FUNCTION_BLOCK FB_MotionInterlocksLimSw IMPLEMENTS I_MotionInterlocks
VAR_INPUT
END_VAR
VAR_OUTPUT
END_VAR
VAR
    iMotionInterlocksCommon : I_MotionInterlocksCommon;
    iLimSwStatus : I_LimSwStatus;
    bError : BOOL;
    nErrorID:UDINT;
    sMessage : T_MAXSTRING;
    {attribute 'hide'}
    bNewMoveReq : BOOL;
    {attribute 'hide'}
    bEnable	: BOOL;
    {attribute 'hide'}
    bReset : BOOL;
    {attribute 'hide'}
    bMoveOk : BOOL;
    bMoveBackwardEnabled : BOOL;
    bMoveForwardEnabled  : BOOL;
    bPowerEnable : BOOL;
    Enable: BOOL;
    {attribute 'hide'}
    bLimHit : BOOL;
    {attribute 'hide'}
    ftForwardEnabled : F_TRIG;
    {attribute 'hide'}
    ftBackwardEnabled : F_TRIG;
    {attribute 'hide'}
    rtUserExec : R_TRIG;
    {attribute 'hide'}
    rtReset : R_TRIG;
    {attribute 'hide'}
    bLimHitIdling : BOOL;
    {attribute 'hide'}
    bLimHitMoving : BOOL;
    {attribute 'hide'}
    bWarning: BOOL;
    {attribute 'hide'}
    bPositiveDirection : BOOL;
    {attribute 'hide'}
    bNegativeDirection : BOOL;
    {attribute 'hide'}
    bHomeBusy : BOOL;
END_VAR

// Read Limits status and update shared space
bMoveBackwardEnabled := THIS^.iLimSwStatus.MoveBackwardEnabled;
bMoveForwardEnabled := THIS^.iLimSwStatus.MoveForwardEnabled;

rtReset(CLK:=bReset);
rtUserExec (CLK:=bNewMoveReq);
ftForwardEnabled(CLK:=bMoveForwardEnabled);
ftBackwardEnabled (CLK:=bMoveBackwardEnabled);

IF NOT THIS^.bHomeBusy AND ((ftForwardEnabled.Q AND THIS^.bPositiveDirection)
        OR (ftBackwardEnabled.Q AND THIS^.bNegativeDirection))THEN
    // Not an error, just a warning
    IF NOT bMoveForwardEnabled THEN
            THIS^.sMessage:='Cannot move past Positive limit.';
    ELSIF NOT bMoveBackwardEnabled THEN
            THIS^.sMessage:='Cannot move past Negative limit.';
    END_IF
    THIS^.bWarning:=TRUE;
    THIS^.bLimHit := TRUE;
    THIS^.bLimHitMoving:=TRUE;
ELSIF rtUserExec.Q OR rtReset.Q THEN
    THIS^.bLimHit := FALSE;
    THIS^.bLimHitMoving := bLimHit;
    THIS^.bLimHitIdling := bLimHit;
    THIS^.sMessage := '';
    THIS^.bWarning := FALSE;
END_IF


IF THIS^.iMotionInterlocksCommon.Error THEN
    bError := THIS^.iMotionInterlocksCommon.Error;
    nErrorID := THIS^.iMotionInterlocksCommon.ErrorID;
    sMessage := THIS^.iMotionInterlocksCommon.Message;
END_IF

PROPERTY Aborted : BOOL
GET
END_GET
END_PROPERTY

PROPERTY Active : BOOL
GET
END_GET
END_PROPERTY

METHOD AxisStatus
VAR_INPUT
    HomeBusy	: BOOL;
    PositiveDirection	: BOOL;
    NegativeDirection	: BOOL;
END_VAR
THIS^.bPositiveDirection := PositiveDirection;
THIS^.bNegativeDirection := NegativeDirection;
THIS^.bHomeBusy := HomeBusy;
END_METHOD

PROPERTY Busy : BOOL
GET
END_GET
END_PROPERTY

METHOD PUBLIC CallAfterInit
VAR_INPUT
    iMotionInterlocksCommon : I_MotionInterlocksCommon;
    iLimSwStatus : I_LimSwStatus;
END_VAR
THIS^.iMotionInterlocksCommon := iMotionInterlocksCommon;
THIS^.iLimSwStatus := iLimSwStatus;
END_METHOD

PROPERTY Done : BOOL
GET
END_GET
END_PROPERTY

METHOD DriveCommands
VAR_INPUT
    Enable	: BOOL;
    NewMoveReq	: BOOL;
    Reset	: BOOL;
END_VAR
bReset :=  Reset;
// Forward drive cmds to Generic interlocks and lim status FB
THIS^.iMotionInterlocksCommon.DriveCommands(Enable:=Enable, NewMoveReq:=NewMoveReq, Reset:=Reset);
END_METHOD

PROPERTY Error : BOOL
GET
Error := bError;
END_GET
END_PROPERTY

PROPERTY ErrorID : UDINT
GET
ErrorID := nErrorID;
END_GET
END_PROPERTY

//FB_Init is always available implicitly and it is used primarily for initialization.
//The return value is not evaluated. For a specific influence, you can also declare the
//methods explicitly and provide additional code there with the standard initialization
//code. You can evaluate the return value.
METHOD FB_Init: BOOL
VAR_INPUT
    bInitRetains: BOOL; // TRUE: the retain variables are initialized (reset warm / reset cold)
    bInCopyCode: BOOL;  // TRUE: the instance will be copied to the copy code afterward (online change)
    iMotionInterlocksCommon : I_MotionInterlocksCommon;
    iLimSwStatus : I_LimSwStatus;
END_VAR
THIS^.iMotionInterlocksCommon  := iMotionInterlocksCommon ;
THIS^.iLimSwStatus := iLimSwStatus;
END_METHOD

PROPERTY InterlockEvent : BOOL
GET
InterlockEvent := THIS^.bLimHit;
END_GET
END_PROPERTY

PROPERTY LimHit : BOOL
GET
Limhit := THIS^.bLimHit;
END_GET
END_PROPERTY

PROPERTY LimHome : BOOL
GET
LimHome := THIS^.iLimSwStatus.LimHome;
END_GET
END_PROPERTY

PROPERTY Message : T_MAXSTRING
GET
Message := sMessage;
END_GET
END_PROPERTY

PROPERTY MoveBackwardEnabled : BOOL
GET
MoveBackwardEnabled := THIS^.iLimSwStatus.MoveBackwardEnabled;
END_GET
END_PROPERTY

PROPERTY MoveForwardEnabled : BOOL
GET
MoveForwardEnabled := THIS^.iLimSwStatus.MoveForwardEnabled;
END_GET
END_PROPERTY

PROPERTY MoveOk : BOOL
GET
MoveOk := THIS^.iMotionInterlocksCommon.MoveOk;
END_GET
END_PROPERTY

PROPERTY PowerEnabled : BOOL
GET
PowerEnabled := THIS^.iMotionInterlocksCommon.PowerEnabled;
END_GET
END_PROPERTY

PROPERTY Warning : BOOL
GET
Warning := THIS^.bWarning;
END_GET
END_PROPERTY

END_FUNCTION_BLOCK

(* stored: Version 1.1.0.1
   POU FB_MotionInterlocksLimSw: Id {158cbb88-3b97-40e2-97dc-4d7a82a1299f}, SpecialFunc None
   Property Aborted: Id {a1175752-7c2c-4d2c-b0ac-3a4f9f39a027}
   Get Get: Id {972c3d12-c93b-46d8-adca-4ce3ce1b4165}
   Property Active: Id {3b34c057-b1ec-4bc7-83b1-4a80ec87a88b}
   Get Get: Id {0ccb4185-7643-4a8c-bdd0-04e775e1ac39}
   Method AxisStatus: Id {6d21d504-ee18-4457-abef-61e8d5df9058}
   Property Busy: Id {a6daac7c-9df9-4ab9-ad3d-28aaab54bf26}
   Get Get: Id {5a6e7c19-94f7-4fad-a884-0cab68944ddd}
   Method CallAfterInit: Id {04046040-41be-4ab4-ade8-8cbc22051e82}
   Property Done: Id {f89b31f3-ca38-4979-a504-0096d2187a3b}
   Get Get: Id {a79d952f-6f18-4524-bb34-0541fc9c86b9}
   Method DriveCommands: Id {61a4eb92-408d-4d90-8d81-bc9594431b56}
   Property Error: Id {e499cdfd-969f-4051-8215-bd6b1edef6bb}
   Get Get: Id {7238505b-9b6a-43fb-ba12-674778d8c8ff}
   Property ErrorID: Id {9d2ee520-34ec-43b6-bfa3-0b9c47c94f72}
   Get Get: Id {a73c59e2-e172-4b19-8c08-958487d94121}
   Method FB_Init: Id {a7a90e7d-0c0f-4077-b585-b6d1f8caabad}
   Property InterlockEvent: Id {1b30ac20-f930-48f6-8ea2-fc10757db2a2}
   Get Get: Id {b809f3cc-6e7f-4e61-b45d-cf84d0c8cc87}
   Property LimHit: Id {616009f9-19f9-42ea-8b14-b1761f35e869}
   Get Get: Id {b3896752-cee8-4d8e-b9d2-857fe8348810}
   Property LimHome: Id {6c566142-67f9-43df-8e4b-bb59f6a41f69}
   Get Get: Id {094be525-7bad-4a92-b899-3a12a85229d6}
   Property Message: Id {6b1916c5-039a-4cea-99b5-b8f805042945}
   Get Get: Id {a8ad55da-d47a-4037-a50e-076da5305f40}
   Property MoveBackwardEnabled: Id {b178f46f-0443-44d6-a91f-16b15ef2cae5}
   Get Get: Id {a268efd3-4ad6-49eb-932a-a234343d2af7}
   Property MoveForwardEnabled: Id {faed5261-6d75-4261-803b-7f0e96c07091}
   Get Get: Id {b3fa4ff6-04dc-4a45-b2b8-d5535c7132d2}
   Property MoveOk: Id {7e64ea4a-5623-4e42-ad55-52145a4215f0}
   Get Get: Id {bb84aff3-ebbf-450c-8040-87d9eb667555}
   Property PowerEnabled: Id {9511d4c7-e78d-40e2-9d5a-6ecffc43a003}
   Get Get: Id {69aad844-8aea-4c31-a561-377909ac709b}
   Property Warning: Id {d4f46c69-4dc7-45e7-9978-5602afa06ae3}
   Get Get: Id {98755ed6-4331-4fcd-ab91-87a47d6bca9e} *)
